// TIA Portal V16 export
// export: Created 2024-12-03T15:41:44.4623272Z, ExportSetting WithDefaults, DisplayName Totally Integrated Automation Portal, DisplayVersion V16 Update 6, DisplayName TIA Portal Version Control Interface, DisplayVersion V16 Update 2, DisplayName TIA Portal Openness, DisplayVersion V16 Update 6, DisplayName TIA Portal Teamcenter Gateway, DisplayVersion V16, DisplayName SINAMICS Startdrive Advanced, DisplayVersion V16 Update 5, DisplayName SINAMICS Startdrive G130, G150, S120, S150, SINAMICS MV, S210, DisplayVersion V16 Update 5, DisplayName SINAMICS Startdrive G110M, G120, G120C, G120D, G120P, G115D, DisplayVersion V16 Update 5, DisplayName STEP 7 Professional, DisplayVersion V16 Update 6, DisplayName STEP 7 Safety, DisplayVersion V16, DisplayName WinCC Advanced / Unified PC, DisplayVersion V16 Update 6
DATA_BLOCK "HMI_DB"   // DB46
{ S7_Optimized_Access := 'FALSE' }
VERSION : 0.1
// stored: AutoNumber true, DBAccessibleFromOPCUA true, IsOnlyStoredInLoadMemory false, IsWriteProtectedInAS false
   VAR
      ResetFromHMI : Bool;
      ResetCounters : "HandShake_UDT";
      RemoveManualOverride : "HandShake_UDT";
      ReloadSettings { S7_SetPoint := 'True'} : "HandShake_UDT";
      SetDefaultTrackings { S7_SetPoint := 'True'} : "HandShake_UDT";
      ResetSensorCounters { S7_SetPoint := 'True'} : "HandShake_UDT";
      WakeUpSignal { S7_SetPoint := 'True'} : Bool;
   END_VAR
BEGIN
END_DATA_BLOCK
